// Mitsubishi GX Works2 project: project (1)   PLC: FX3G

// global labels: Global1
VAR_GLOBAL
  Start_day AT X007 : BOOL;
  Bisquit_Q AT D1101 : INT;
  Cream_Q AT D1105 : INT;
  Chocolate_Q AT D1109 : INT;
END_VAR
VAR_GLOBAL CONSTANT
  Bisquit_Min : INT := 6;
  Cream_Min : INT := 300;
  Chocolate_Min : INT := 240;
END_VAR
VAR_GLOBAL
  Sys_On AT Y007 : BOOL;
  Start_cream AT X011 : BOOL;
END_VAR
VAR_GLOBAL CONSTANT
  Bisquit_minus : INT := 6;
  Cream_minus : INT := 300;
END_VAR
VAR_GLOBAL
  input_bisquit AT D1140 : INT;
  input_cream AT D1143 : INT;
  input_chocolate AT D1146 : INT;
  endDay AT M9 : BOOL;
  endDayZero AT M28 : BOOL;
  Day_over AT Y006 : BOOL;
  Dddddd AT M52 : BOOL;
  cfga AT M52 : BOOL;
  mfgk AT X010 : BOOL;
  dgsd AT X010 : BOOL;
  move_to_B AT M2 : BOOL;
  Stop_blink AT M5 : BOOL;
  monitir_lighter AT M3 : BOOL;
  end_blink AT TS1 : BOOL;
  blink0 AT Y000 : BOOL;
  end_blink2 AT TS2 : BOOL;
  blink1 AT Y001 : BOOL;
END_VAR
VAR_GLOBAL CONSTANT
  time_blink1 : INT := 10;
  time_blink : INT := 10;
  time_blink2 : INT := 10;
END_VAR
VAR_GLOBAL
  timer_blink2 AT TC2 : BOOL;
  timer_blink1 AT TC1 : BOOL;
  Start_blink AT M0 : BOOL;
  counter_seconds AT TC3 : BOOL;
END_VAR
VAR_GLOBAL CONSTANT
  timer_4sec : INT := 40;
END_VAR
VAR_GLOBAL
  count4_sec AT TS3 : BOOL;
  Start_machineA AT X010 : BOOL;
  machineA_on AT M6 : BOOL;
  Sen_krembo AT X002 : BOOL;
  sen_30 AT X003 : BOOL;
  sen_cam AT X004 : BOOL;
  emergency AT X005 : BOOL;
  sen_15 AT X001 : BOOL;
  cream_on AT Y004 : BOOL;
END_VAR
VAR_GLOBAL CONSTANT
  Double_chocolate : INT := 240;
  chocolate : INT := 120;
END_VAR
VAR_GLOBAL
  machineB_on AT X006 : BOOL;
  analog_input_1 AT D8280 : INT;
END_VAR
VAR_GLOBAL CONSTANT
  normalization : REAL := 390.0;
END_VAR
VAR_GLOBAL
  Deep_chocolate AT D1115 : REAL;
  saveDeep AT M7 : BOOL;
END_VAR
VAR_GLOBAL CONSTANT
  Double_chocolate_deep : REAL := 5;
END_VAR
VAR_GLOBAL
  finishDeep AT Y003 : BOOL;
  timer_Deep AT TC4 : BOOL;
END_VAR
VAR_GLOBAL CONSTANT
  time_deep : INT := 50;
END_VAR
VAR_GLOBAL
  pack AT X000 : BOOL;
END_VAR
VAR_GLOBAL CONSTANT
  krembo_5 : INT := 5;
END_VAR
VAR_GLOBAL
  counter_krembo AT CC1 : BOOL;
  Last_krembo AT Y002 : BOOL;
  down_counter_krembo AT CS1 : BOOL;
  counter_krembo_close AT CC2 : BOOL;
END_VAR
VAR_GLOBAL CONSTANT
  krembo_6 : INT := 6;
END_VAR
VAR_GLOBAL
  down_counter_krembo6 AT CS2 : BOOL;
  sum_krembo AT D1120 : REAL;
END_VAR
VAR_GLOBAL CONSTANT
  krembo_inf : INT := 10000;
  normalization2 : REAL := 40.8;
END_VAR
VAR_GLOBAL
  analogOutput AT D1198 : REAL;
  analog_output AT D8282 : INT;
  blink3SEC AT M39 : BOOL;
END_VAR
VAR_GLOBAL CONSTANT
  timer_3sec : INT := 30;
END_VAR
VAR_GLOBAL
  Stop_blink_End AT M35 : BOOL;
  monitir_lighter_end AT M3 : BOOL;
  timer_blink1_end AT TC5 : BOOL;
  end_blink_end AT TS5 : BOOL;
  monitir_lighter_end_end AT M33 : BOOL;
  timer_blink2_end AT TC6 : BOOL;
  end_blink2_end AT TS6 : BOOL;
  counter_seconds_end AT TC11 : BOOL;
  counter_4seconds_end AT TS11 : BOOL;
  Sys_OnCheck AT Y011 : BOOL;
  ziluf_cream AT D1150 : INT;
  tvila_chocolate AT D1155 : INT;
END_VAR

// task Task_01 (event TRUE, interval 0, priority 31): POU_01

PROGRAM POU_01
VAR CONSTANT
  plus_1 : REAL := 1;
END_VAR
(* structured ladder/FBD written out as ST: instructions are called as NAME(EN, inputs, outputs); _pN, _eN, _tN stand for wires *)
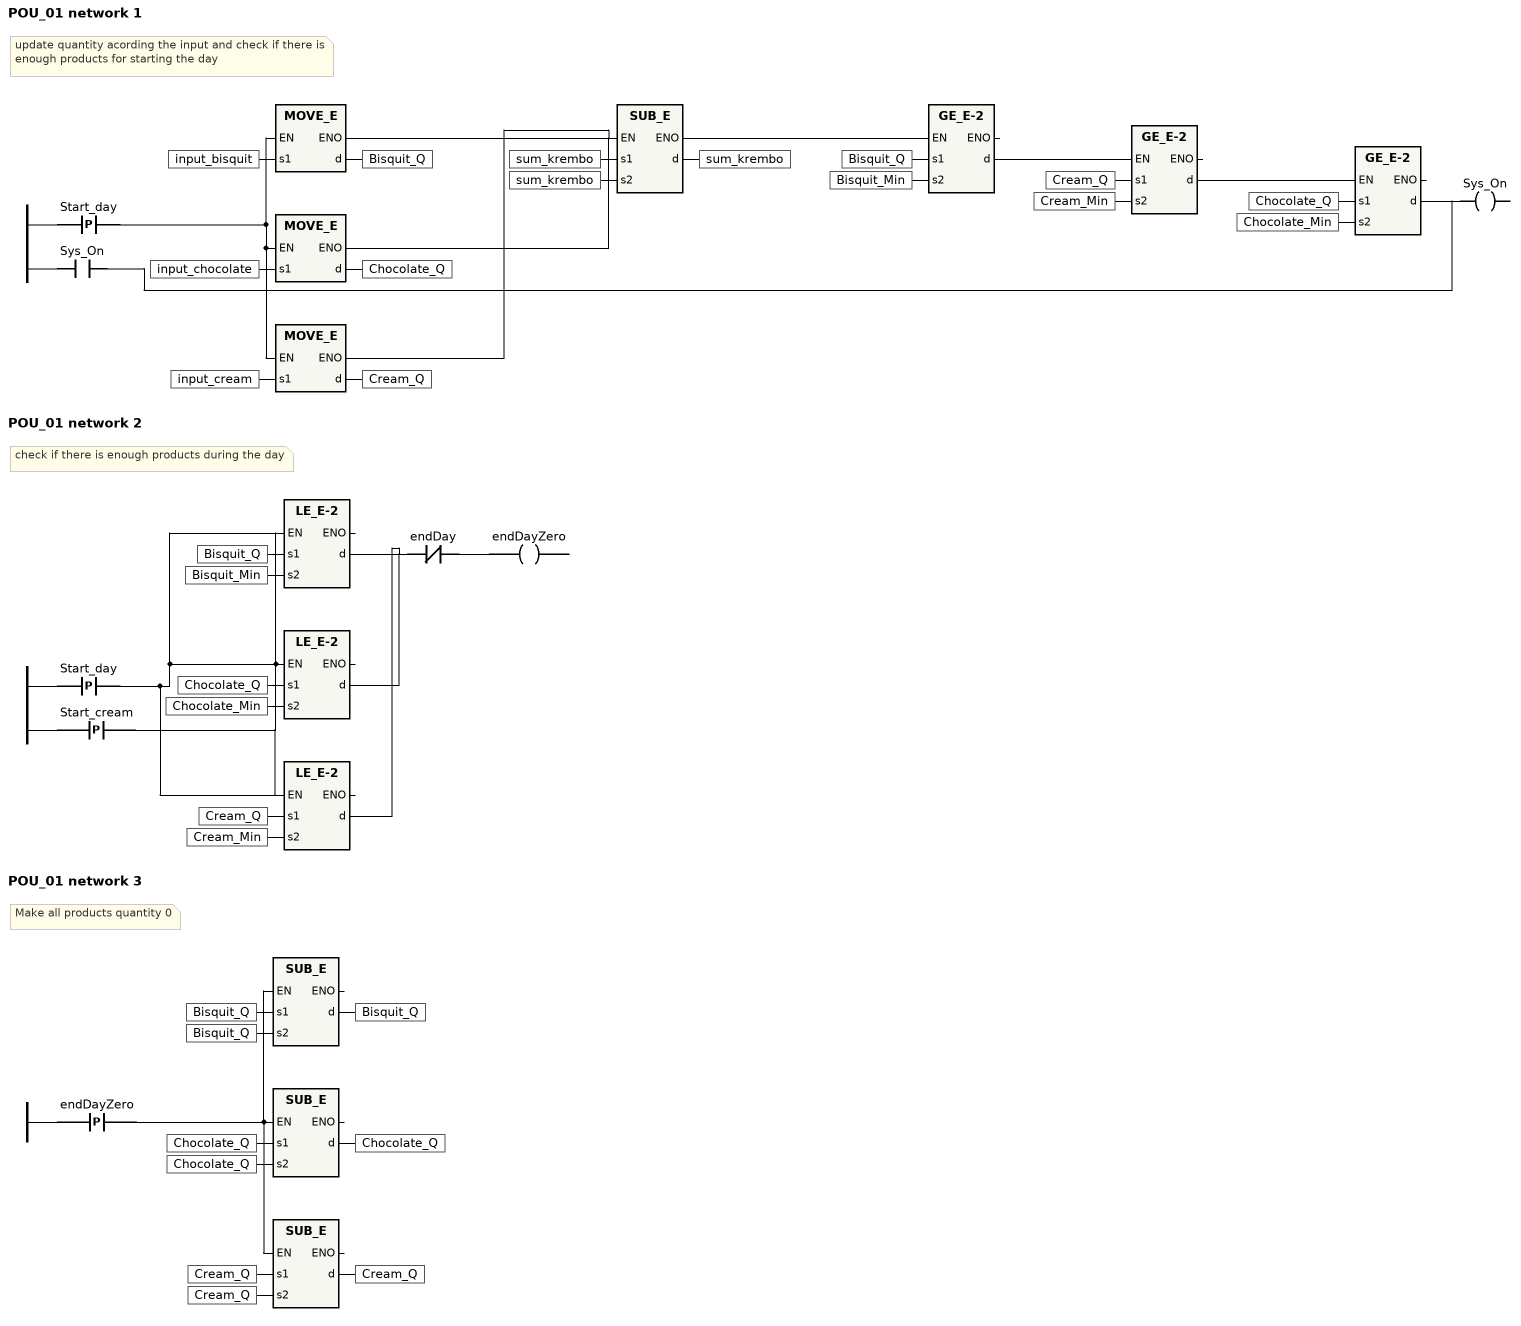
(* network 1 *)
(* update quantity acording the input and check if there is enough products for starting the day *)
_p1 := LDP(TRUE, Start_day);
_e2 := MOVE_E(_p1, input_bisquit, Bisquit_Q);
_e3 := MOVE_E(_p1, input_chocolate, Chocolate_Q);
_e4 := MOVE_E(_p1, input_cream, Cream_Q);
_e5 := SUB_E(_e2 OR _e3 OR _e4, sum_krembo, sum_krembo, sum_krembo);
GE_E(_e5, Bisquit_Q, Bisquit_Min, _t6);
GE_E(_t6, Cream_Q, Cream_Min, _t7);
GE_E(_t7, Chocolate_Q, Chocolate_Min, _t8);
Sys_On := _t8 OR Sys_On;
(* network 2 *)
(* check if there is enough products during the day *)
_p1 := LDP(TRUE, Start_day) OR LDP(TRUE, Start_cream);
LE_E(_p1, Bisquit_Q, Bisquit_Min, _t2);
LE_E(_p1, Chocolate_Q, Chocolate_Min, _t3);
LE_E(_p1, Cream_Q, Cream_Min, _t4);
endDayZero := (_t2 OR _t3 OR _t4) AND NOT endDay;
(* network 3 *)
(* Make all products quantity 0 *)
_p1 := LDP(TRUE, endDayZero);
SUB_E(_p1, Bisquit_Q, Bisquit_Q, Bisquit_Q);
SUB_E(_p1, Chocolate_Q, Chocolate_Q, Chocolate_Q);
SUB_E(_p1, Cream_Q, Cream_Q, Cream_Q);
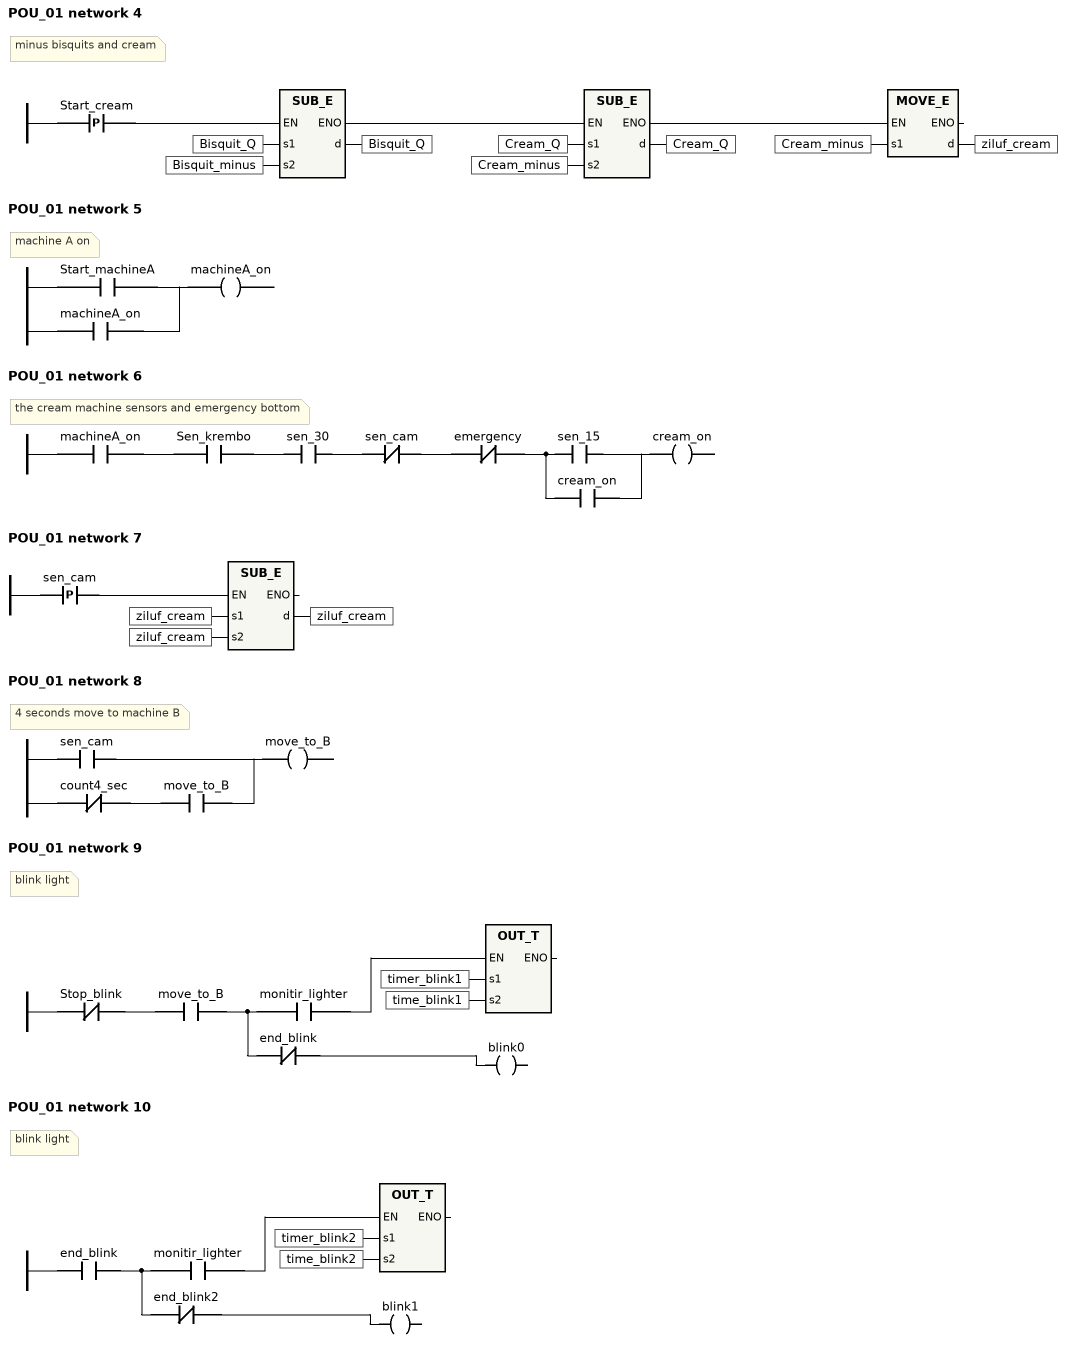
(* network 4 *)
(* minus bisquits and cream *)
_e1 := SUB_E(LDP(TRUE, Start_cream), Bisquit_Q, Bisquit_minus, Bisquit_Q);
_e2 := SUB_E(_e1, Cream_Q, Cream_minus, Cream_Q);
MOVE_E(_e2, Cream_minus, ziluf_cream);
(* network 5 *)
(* machine A on *)
machineA_on := Start_machineA OR machineA_on;
(* network 6 *)
(* the cream machine sensors and emergency bottom *)
_p1 := machineA_on AND Sen_krembo AND sen_30 AND NOT sen_cam AND NOT emergency;
cream_on := (_p1 AND sen_15) OR (_p1 AND cream_on);
(* network 7 *)
SUB_E(LDP(TRUE, sen_cam), ziluf_cream, ziluf_cream, ziluf_cream);
(* network 8 *)
(* 4 seconds move to machine B *)
move_to_B := sen_cam OR (NOT count4_sec AND move_to_B);
(* network 9 *)
(* blink light *)
_p1 := NOT Stop_blink AND move_to_B;
OUT_T(_p1 AND monitir_lighter, timer_blink1, time_blink1);
blink0 := _p1 AND NOT end_blink;
(* network 10 *)
(* blink light *)
OUT_T(end_blink AND monitir_lighter, timer_blink2, time_blink2);
blink1 := end_blink AND NOT end_blink2;
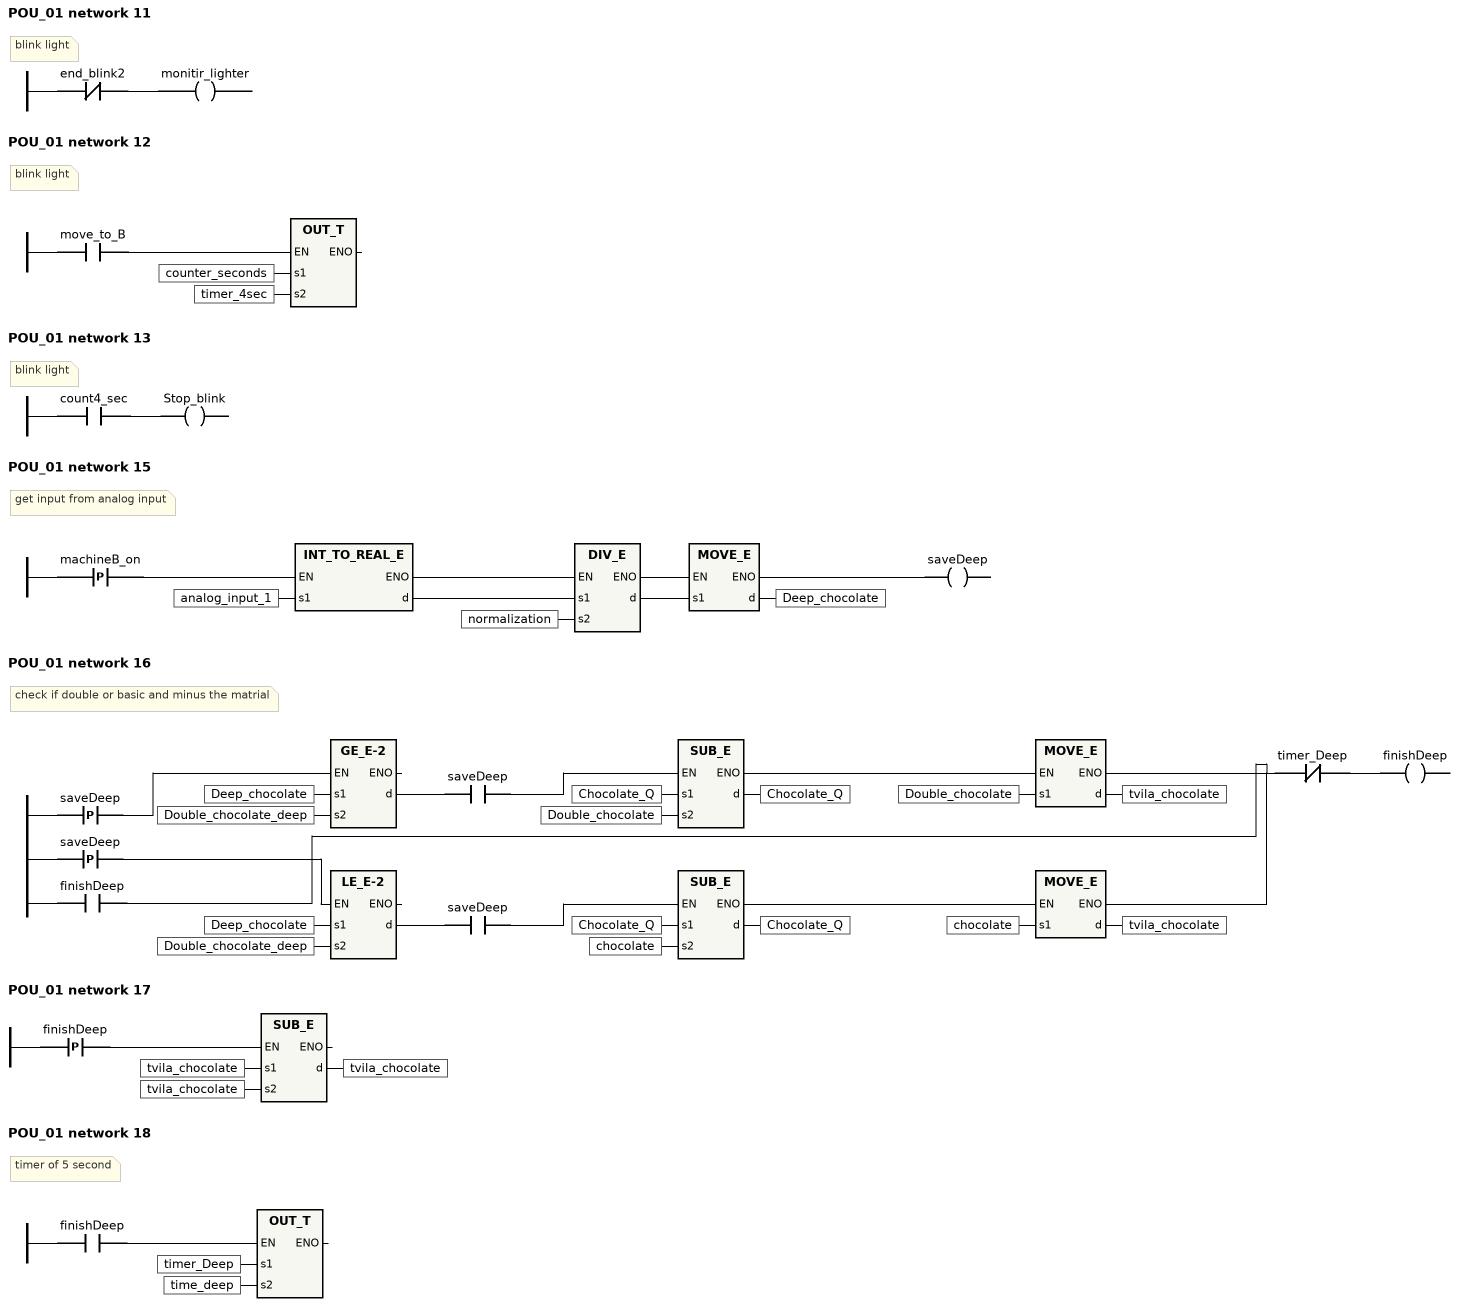
(* network 11 *)
(* blink light *)
monitir_lighter := NOT end_blink2;
(* network 12 *)
(* blink light *)
OUT_T(move_to_B, counter_seconds, timer_4sec);
(* network 13 *)
(* blink light *)
Stop_blink := count4_sec;
(* network 15 *)
(* get input from analog input *)
_e2 := INT_TO_REAL_E(LDP(TRUE, machineB_on), analog_input_1, _t1);
_e4 := DIV_E(_e2, _t1, normalization, _t3);
_e5 := MOVE_E(_e4, _t3, Deep_chocolate);
saveDeep := _e5;
(* network 16 *)
(* check if double or basic and minus the matrial *)
GE_E(LDP(TRUE, saveDeep), Deep_chocolate, Double_chocolate_deep, _t1);
_e2 := SUB_E(_t1 AND saveDeep, Chocolate_Q, Double_chocolate, Chocolate_Q);
_e3 := MOVE_E(_e2, Double_chocolate, tvila_chocolate);
LE_E(LDP(TRUE, saveDeep), Deep_chocolate, Double_chocolate_deep, _t4);
_e5 := SUB_E(_t4 AND saveDeep, Chocolate_Q, chocolate, Chocolate_Q);
_e6 := MOVE_E(_e5, chocolate, tvila_chocolate);
finishDeep := (_e3 OR _e6 OR finishDeep) AND NOT timer_Deep;
(* network 17 *)
SUB_E(LDP(TRUE, finishDeep), tvila_chocolate, tvila_chocolate, tvila_chocolate);
(* network 18 *)
(* timer of 5 second *)
OUT_T(finishDeep, timer_Deep, time_deep);
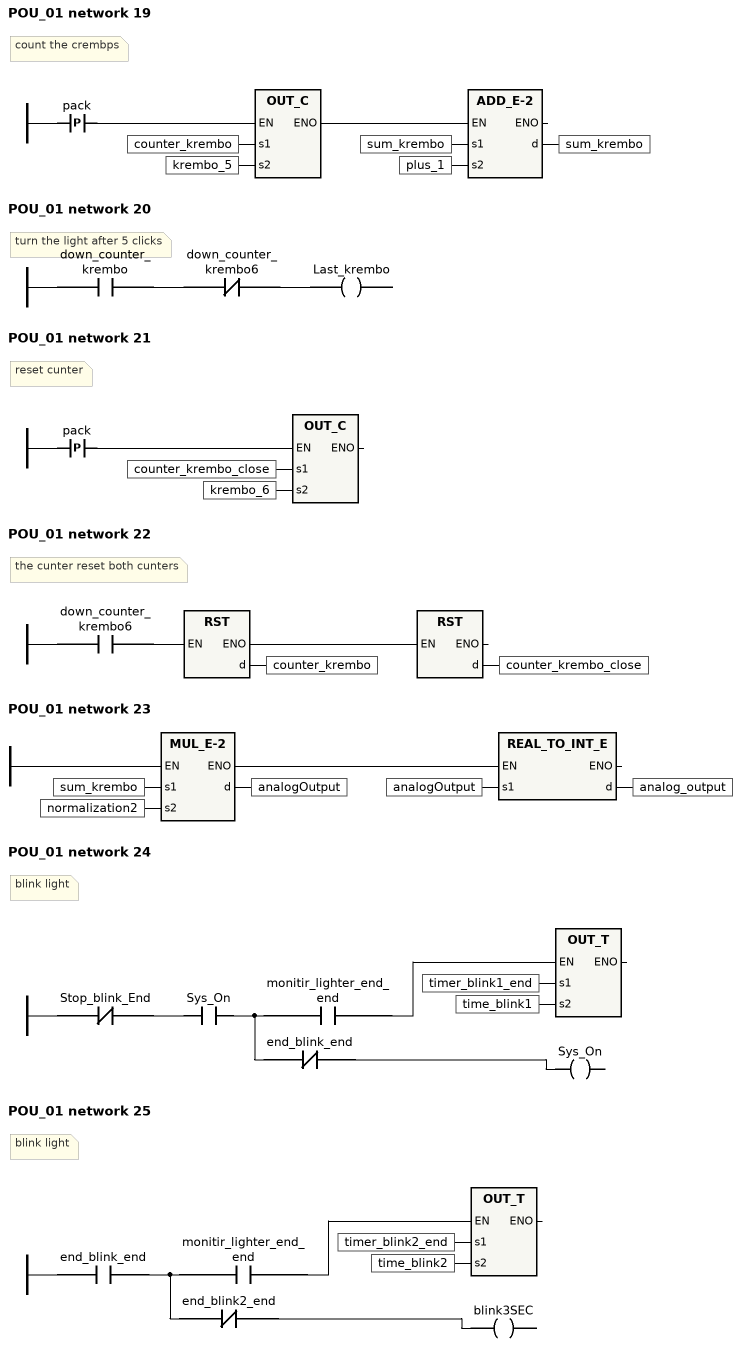
(* network 19 *)
(* count the crembps *)
_e1 := OUT_C(LDP(TRUE, pack), counter_krembo, krembo_5);
ADD_E(_e1, sum_krembo, plus_1, sum_krembo);
(* network 20 *)
(* turn the light after 5 clicks *)
Last_krembo := down_counter_krembo AND NOT down_counter_krembo6;
(* network 21 *)
(* reset cunter *)
OUT_C(LDP(TRUE, pack), counter_krembo_close, krembo_6);
(* network 22 *)
(* the cunter reset both cunters *)
_e1 := RST(down_counter_krembo6, counter_krembo);
RST(_e1, counter_krembo_close);
(* network 23 *)
_e1 := MUL_E(TRUE, sum_krembo, normalization2, analogOutput);
REAL_TO_INT_E(_e1, analogOutput, analog_output);
(* network 24 *)
(* blink light *)
_p1 := NOT Stop_blink_End AND Sys_On;
OUT_T(_p1 AND monitir_lighter_end_end, timer_blink1_end, time_blink1);
Sys_On := _p1 AND NOT end_blink_end;
(* network 25 *)
(* blink light *)
OUT_T(end_blink_end AND monitir_lighter_end_end, timer_blink2_end, time_blink2);
blink3SEC := end_blink_end AND NOT end_blink2_end;
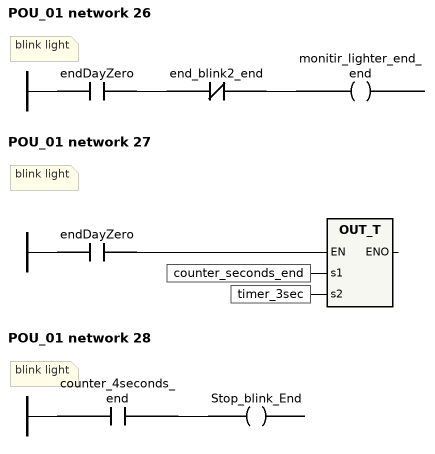
(* network 26 *)
(* blink light *)
monitir_lighter_end_end := endDayZero AND NOT end_blink2_end;
(* network 27 *)
(* blink light *)
OUT_T(endDayZero, counter_seconds_end, timer_3sec);
(* network 28 *)
(* blink light *)
Stop_blink_End := counter_4seconds_end;
END_PROGRAM
